RoboDK station: smart_factory.rdk

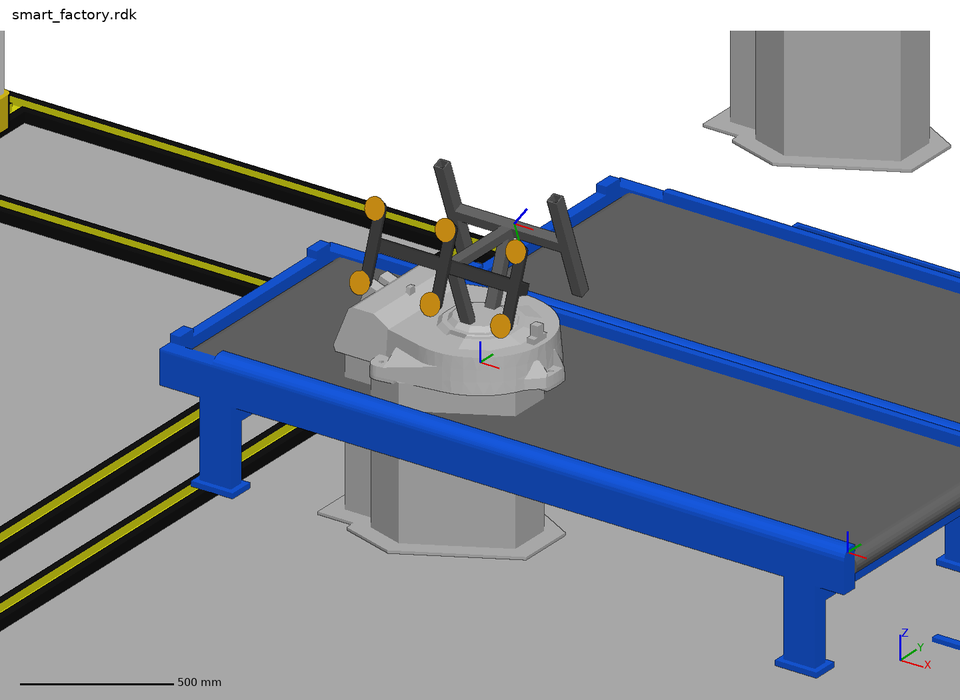
[picture v0: the station drawn from its stored meshes, robots at their saved joint values, targets as dots, program paths as lines]
Station smart_factory (saved by RoboDK 5.9.0). Poses are relative to the parent item; angles as X-Y-Z fixed-axis rotations.
  - frame Main_Frame at (0, 0, 0) mm
    - folder Rack
      - frame Rack1 Base at (-5000, 1000, 50) mm, rotated rx 0 ry 0 rz -90 deg
        - robot Rack1: 2 axes
            modified DH rows (alpha deg, a mm, theta deg, d mm): 0, 0, 0, 0 linear; 90, 0, 0, 0 linear
            base shift (0, 0, 0) mm, rotated rx 0 ry 90 rz 0 deg
            joint limits [-3250, -2100] to [0, 0]; home [0, 0]; saved at [0, 0]
      - frame Rack2 Base at (-5000, 1000, 50) mm, rotated rx 0 ry 0 rz -90 deg
        - robot Rack2: 2 axes
            modified DH rows (alpha deg, a mm, theta deg, d mm): 0, 0, 0, 0 linear; 90, 0, 0, 0 linear
            base shift (0, 0, 0) mm, rotated rx 0 ry 90 rz 0 deg
            joint limits [-3250, -2100] to [0, 0]; home [0, 0]; saved at [-1000, 0]
      - frame Rack3 Base at (-5000, 1000, 50) mm, rotated rx 0 ry 0 rz -90 deg
        - robot Rack3: 2 axes
            modified DH rows (alpha deg, a mm, theta deg, d mm): 0, 0, 0, 0 linear; 90, 0, 0, 0 linear
            base shift (0, 0, 0) mm, rotated rx 0 ry 90 rz 0 deg
            joint limits [-3250, -2100] to [0, 0]; home [0, 0]; saved at [-2000, 0]
      - frame Rack4 Base at (-5000, 1000, 50) mm, rotated rx 0 ry 0 rz -90 deg
        - robot Rack4: 2 axes
            modified DH rows (alpha deg, a mm, theta deg, d mm): 0, 0, 0, 0 linear; 90, 0, 0, 0 linear
            base shift (0, 0, 0) mm, rotated rx 0 ry 90 rz 0 deg
            joint limits [-3250, -2100] to [0, 0]; home [0, 0]; saved at [-3000, 0]
    - object Room at (0, 0, 0) mm, size 10000 x 10000 x 25 mm, geometry from Room.stl
    - folder Conveyor
      - frame CON1 Base at (450, 4000, 500) mm
        - robot CON1: 1 axes
            modified DH rows (alpha deg, a mm, theta deg, d mm): 0, 0, 0, 0 linear
            base shift (0, 0, 0) mm, rotated rx 0 ry 90 rz 0 deg
            joint limits [-200000] to [200000]; home [0]; saved at [0]
      - frame CON2 Base at (530, 4850, 500) mm, rotated rx 0 ry 0 rz -180 deg
        - robot CON2: 1 axes
            modified DH rows (alpha deg, a mm, theta deg, d mm): 0, 0, 0, 0 linear
            base shift (0, 0, 0) mm, rotated rx 0 ry 90 rz 0 deg
            joint limits [-200000] to [200000]; home [0]; saved at [0]
    - frame Robot1_Main_Frame at (-1800, 1300, 0) mm
      - object Robot1_Base at (0, 1990, 50) mm, size 751 x 658 x 590 mm, geometry from R1_BASE.stl
      - frame ABB1 Base at (129.07, 2001.45, 640) mm
        - robot ABB1 (model ABB IRB 2400/16): 6 axes, payload 16 kg, reach 1550 mm, repeatability 0.03 mm, weight 380 kg
            joint limits [-180, -100, -60, -200, -120, -400] to [180, 110, 65, 200, 120, 400]; home [0, 0, 0, 0, 0, 0]; saved at [90, 30, 50, 90, 0, -90]
          - tool ABB1_T, TCP at (0, 0, 200) mm
          - frame ABB1_TR Base at (0, 195, 425) mm, rotated rx -70 ry 0 rz 0 deg
            - robot ABB1_TR: 1 axes
                joint limits [-20] to [200]; home [0]; saved at [100]
        - object Robot1_Base at (0, 1990, 50) mm, size 751 x 658 x 590 mm, geometry from R1_BASE.stl
  - Python program Prog1 (listed below)
  - frame CON3 Base at (0, 3000, 540) mm
    - robot CON3: 1 axes
        modified DH rows (alpha deg, a mm, theta deg, d mm): 0, 0, 0, 0 linear
        base shift (0, 0, 0) mm, rotated rx 0 ry 90 rz 0 deg
        joint limits [-200000] to [200000]; home [0]; saved at [0]
  - frame CON4 Base at (0, 4000, 0) mm
    - robot CON4: 1 axes
        modified DH rows (alpha deg, a mm, theta deg, d mm): 0, 0, 0, 0 linear
        base shift (0, 0, 0) mm, rotated rx 0 ry 90 rz 0 deg
        joint limits [-200000] to [200000]; home [0]; saved at [0]
  - frame CON5 Base at (0, 5000, 0) mm
    - robot CON5: 1 axes
        modified DH rows (alpha deg, a mm, theta deg, d mm): 0, 0, 0, 0 linear
        base shift (0, 0, 0) mm, rotated rx 0 ry 90 rz 0 deg
        joint limits [0] to [970]; home [0]; saved at [0]

--- Python program Prog1 ---
from robodk import robolink    # RoboDK API
from robodk import robomath    # Robot toolbox
RDK = robolink.Robolink()

from robodk import *      # RoboDK API
from robolink import *    # Robot toolbox

Rack1 = RDK.Item("Rack1", 2)
Rack2 = RDK.Item("Rack2", 2)
Rack3 = RDK.Item("Rack3", 2)
Rack4 = RDK.Item("Rack4", 2)

Main_Frame = RDK.Item("Main_Frame", 3)
Rack1_Frame = RDK.Item("Rack1 Base", 3)
Rack2_Frame = RDK.Item("Rack2 Base", 3)
Rack3_Frame = RDK.Item("Rack3 Base", 3)
Rack4_Frame = RDK.Item("Rack4 Base", 3)

Room = RDK.Item("Room", 5)

def parse_matrix(matrix_str):
    lines = matrix_str.strip().split('\n')
    matrix = []
    for line in lines:
        line = line.strip().strip(';').strip('[]')  # [, ], ; 제거
        values = line.split(',')
        row = [float(val.strip()) for val in values]
        matrix.append(row)
    return matrix

def reset1():
    p1 = parse_matrix("""[     1.000000,     0.000000,     0.000000,     0.000000 ;
        0.000000,     1.000000,     0.000000,     0.000000 ;
        0.000000,     0.000000,     1.000000,     0.000000 ;
        0.000000,     0.000000,     0.000000,     1.000000 ];
    """)
    Room.setParent(Main_Frame)
    Room.setPose(Mat(p1))

    r1 = parse_matrix("""[     0.000000,     1.000000,     0.000000, -5000.000000 ;
        -1.000000,     0.000000,     0.000000,  1000.000000 ;
        0.000000,     0.000000,     1.000000,    50.000000 ;
        0.000000,     0.000000,     0.000000,     1.000000 ];
    """)

    Rack1_Frame.setPose(Mat(r1))
    Rack2_Frame.setPose(Mat(r1))
    Rack3_Frame.setPose(Mat(r1))
    Rack4_Frame.setPose(Mat(r1))

    Rack1_Frame.setParent(Main_Frame)
    Rack2_Frame.setParent(Main_Frame)
    Rack3_Frame.setParent(Main_Frame)
    Rack4_Frame.setParent(Main_Frame)

    Rack1.setParent(Rack1_Frame)
    Rack2.setParent(Rack2_Frame)
    Rack3.setParent(Rack3_Frame)
    Rack4.setParent(Rack4_Frame)


##############################################

CON1 = RDK.Item("CON1", 2)
CON1_Frame = RDK.Item("CON1 Base", 3)
CON2 = RDK.Item("CON2", 2)
CON2_Frame = RDK.Item("CON2 Base", 3)
CON3 = RDK.Item("CON3", 2)
CON3_Frame = RDK.Item("CON3 Base", 3)
CON4 = RDK.Item("CON4", 2)
CON4_Frame = RDK.Item("CON4 Base", 3)
CON5 = RDK.Item("CON5", 2)
CON5_Frame = RDK.Item("CON5 Base", 3)

def reset2():
    con_pos1 = parse_matrix("""[     1.000000,     0.000000,     0.000000,   450.000000 ;
        0.000000,     1.000000,     0.000000,  4000.000000 ;
        0.000000,     0.000000,     1.000000,   500.000000 ;
        0.000000,     0.000000,     0.000000,     1.000000 ];
    """)
    con_pos2 = parse_matrix("""[    -1.000000,     0.000000,     0.000000,   530.000000 ;
        -0.000000,    -1.000000,     0.000000,  4850.000000 ;
        0.000000,     0.000000,     1.000000,   500.000000 ;
        0.000000,     0.000000,     0.000000,     1.000000 ];
    """)

    CON1_Frame.setPose(Mat(con_pos1))
    CON1_Frame.setParent(Main_Frame)
    CON1.setParent(CON1_Frame)

    CON2_Frame.setPose(Mat(con_pos2))
    CON2_Frame.setParent(Main_Frame)
    CON2.setParent(CON2_Frame)

Robot1_Main_Frame = RDK.Item("Robot1_Main_Frame", 3)
Robot1_Base = RDK.Item("Robot1_Base", 5)
ABB1_Base = RDK.Item("ABB1 Base", 3)
ABB1 = RDK.Item("ABB1", 2)
ABB1_Tool_Base = RDK.Item("ABB1_Tool_Base", 3)
ABB1_Tool = RDK.Item("ABB1_Tool", 4)
